PROGRAM test
VAR
	test		:SR;
	Test_1		:R_TRIG;
END_VAR

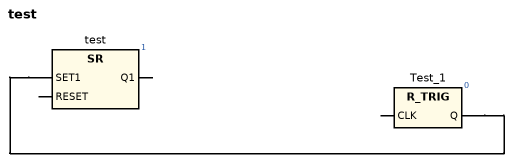
Test_1(); // R_TRIG
test(SET1 := Test_1.Q); // SR

END_PROGRAM

(* stored: Version 1.1.0.1
   POU test: Id {bc63994c-2e25-4bab-a2fc-348711724661}, SpecialFunc None *)
